FUNCTION Convert_LREAL_TO_TIME : Hresult
VAR_INPUT
	in : LREAL;
	out : REFERENCE TO TIME;
END_VAR
VAR
	converted : TIME;
END_VAR
VAR CONSTANT
	INCOMPATIBLE : HRESULT := 16#9811070E;
END_VAR

converted := LREAL_TO_TIME(in);

IF (TIME_TO_LREAL(converted) <> in) THEN
	Convert_LREAL_TO_TIME := INCOMPATIBLE;
	RETURN;
END_IF

out := converted;

END_FUNCTION

(* stored: Version 1.1.0.1, ProductVersion 3.1.4024.12
   POU Convert_LREAL_TO_TIME: Id {b45082cb-a628-4a24-8add-6ffe861eb152}, SpecialFunc None *)
